# B&R Automation Studio project POM_lab1
Automation Studio 4.5.2.102; technology packages: mappMotion 5.2.1

## Configuration labBR

CPU 4PP065.0571-P74, AutomationRuntime D4.52, Build 4.1.2, Vc V4.52.0, Safety 1.10

### Task classes (Cpu.sw)
```
Cyclic#4:
  Program <- Program.prg
Libraries: McBase, MotorCtrl
```

### Hardware
```
4PP065_0571_P74 : 4PP065.0571-P74 v1.1.2.0
  Connector IF5:
    ActivateDevice = 1
    Mode = Manual
    InternetAddress = 10.0.1.10
    SubnetMask = 255.255.255.0
  ConfigurationID = labBR
  Simulation = 1
```

## Logical view

Binary libraries used (declarations not repeated): operator, runtime, astime, AsIecCon, McBase 5.02.1


### Program Logical/Program (ANSIC)

#### Variables.var
```iecst
VAR
	fb_motor : FB_Motor;
	fb_motor_noreg : FB_Motor;
	fb_regulator : FB_Regulator;
	cnt : USINT;
	speed : REAL;
	enable : BOOL;
END_VAR
```

#### Cyclic.c
```c
#include <bur/plctypes.h>

#ifdef _DEFAULT_INCLUDES
	#include <AsDefault.h>
#endif

void _CYCLIC ProgramCyclic(void)
{
	if(enable) {
		speed = 5;
		cnt++;
	} else {
		speed = 0;
	}
	fb_regulator.e = speed - fb_motor.w;
	fb_motor.u = fb_regulator.u * fb_motor.ke;
	fb_motor_noreg.u = speed * fb_motor_noreg.ke;
	FB_Motor(&fb_motor);
	FB_Motor(&fb_motor_noreg);
	FB_Regulator(&fb_regulator);
}
```

#### Init.c
```c
#include <bur/plctypes.h>

#ifdef _DEFAULT_INCLUDES
	#include <AsDefault.h>
#endif

void _INIT ProgramInit(void)
{
	enable = 0;
	cnt = 0;
	speed = 0;

	fb_motor.dt = 0.02;
	fb_motor.ke = 43.98;
	fb_motor.Tm = 0.173;

	fb_motor_noreg.dt = 0.02;
	fb_motor_noreg.ke = 43.98;
	fb_motor_noreg.Tm = 0.173;

	fb_regulator.dt = 0.02;
	fb_regulator.k_p = 2.174;
	fb_regulator.k_i = 12.56;
	fb_regulator.max_abs_value = 24;
}
```

### Library Logical/MotorCtrl (ANSIC)

#### MotorCtrl.fun - Exported functions and function blocks
```iecst
{REDUND_ERROR} {REDUND_UNREPLICABLE} FUNCTION_BLOCK FB_Integrator (*TODO: Add your comment here*) (*$GROUP=User,$CAT=User,$GROUPICON=User.png,$CATICON=User.png*)
	VAR_INPUT
		in : {REDUND_UNREPLICABLE} REAL;
	END_VAR
	VAR_OUTPUT
		out : {REDUND_UNREPLICABLE} REAL;
	END_VAR
	VAR
		dt : {REDUND_UNREPLICABLE} REAL;
	END_VAR
END_FUNCTION_BLOCK

{REDUND_ERROR} {REDUND_UNREPLICABLE} FUNCTION_BLOCK FB_Motor (*TODO: Add your comment here*) (*$GROUP=User,$CAT=User,$GROUPICON=User.png,$CATICON=User.png*)
	VAR_INPUT
		u : {REDUND_UNREPLICABLE} REAL;
	END_VAR
	VAR_OUTPUT
		w : {REDUND_UNREPLICABLE} REAL;
		phi : {REDUND_UNREPLICABLE} REAL;
	END_VAR
	VAR
		integrator : {REDUND_UNREPLICABLE} FB_Integrator;
		Tm : {REDUND_UNREPLICABLE} REAL;
		ke : {REDUND_UNREPLICABLE} REAL;
		dt : {REDUND_UNREPLICABLE} REAL;
		buf : {REDUND_UNREPLICABLE} REAL;
	END_VAR
END_FUNCTION_BLOCK

{REDUND_ERROR} {REDUND_UNREPLICABLE} FUNCTION_BLOCK FB_Regulator (*TODO: Add your comment here*) (*$GROUP=User,$CAT=User,$GROUPICON=User.png,$CATICON=User.png*)
	VAR_INPUT
		e : {REDUND_UNREPLICABLE} REAL;
	END_VAR
	VAR_OUTPUT
		u : {REDUND_UNREPLICABLE} REAL;
	END_VAR
	VAR
		k_p : {REDUND_UNREPLICABLE} REAL;
		k_i : {REDUND_UNREPLICABLE} REAL;
		integrator : {REDUND_UNREPLICABLE} FB_Integrator;
		iyOld : {REDUND_UNREPLICABLE} REAL;
		max_abs_value : {REDUND_UNREPLICABLE} REAL;
		dt : {REDUND_UNREPLICABLE} REAL;
		buf_up : {REDUND_UNREPLICABLE} REAL;
		buf_down : {REDUND_UNREPLICABLE} REAL;
		sum : {REDUND_UNREPLICABLE} REAL;
	END_VAR
END_FUNCTION_BLOCK
```

#### FB_Integrator.c
```c
#include <bur/plctypes.h>
#ifdef __cplusplus
	extern "C"
	{
#endif
	#include "MotorCtrl.h"
#ifdef __cplusplus
	};
#endif
/* TODO: Add your comment here */
void FB_Integrator(struct FB_Integrator* inst)
{
	inst->dt = 0.02;
	inst->out += inst->dt * inst->in;
}
```

#### FB_Motor.c
```c
#include <bur/plctypes.h>
#ifdef __cplusplus
	extern "C"
	{
#endif
	#include "MotorCtrl.h"
#ifdef __cplusplus
	};
#endif
/* TODO: Add your comment here */
void FB_Motor(struct FB_Motor* inst)
{
	/*TODO: Add your code here*/
	inst->buf = (inst->u * (1/inst->ke) - inst->w)*(1/inst->Tm);

	inst->integrator.in = inst->buf;
	FB_Integrator(&inst->integrator);
	inst->w = inst->integrator.out;

	inst->integrator.in = inst->w;
	FB_Integrator(&inst->integrator);
	inst->phi = inst->integrator.out;
}
```

#### FB_Regulator.c
```c
#include <bur/plctypes.h>
#ifdef __cplusplus
	extern "C"
	{
#endif
	#include "MotorCtrl.h"
#ifdef __cplusplus
	};
#endif
/* TODO: Add your comment here */
void FB_Regulator(struct FB_Regulator* inst)
{
	/*TODO: Add your code here*/
	inst->buf_up = inst->e * inst->k_p;
	if(inst->buf_up > inst->max_abs_value || inst->buf_up < -inst->max_abs_value)
	{
		if (inst->buf_up > 0) {
			inst->buf_up = inst->max_abs_value;
		} else if (inst->buf_up < 0){
			inst->buf_up = -inst->max_abs_value;
		}
	}

	inst->buf_down = inst->e * inst->k_i + inst->iyOld;

	inst->integrator.in = inst->buf_down;
	FB_Integrator(&(inst->integrator));
	inst->buf_down = inst->integrator.out;

	inst->sum = inst->buf_up + inst->buf_down;

	if(inst->sum > inst->max_abs_value || inst->sum < -inst->max_abs_value)
	{
		if (inst->sum > 0) {
			inst->sum = inst->max_abs_value;
		} else if (inst->sum < 0) {
			inst->sum = -inst->max_abs_value;
		}
	}
	inst->u = inst->sum;
	inst->iyOld = inst->u - inst->sum;
}
```

Listed in the project but not available here: Logical/Global.var, Logical/Global.typ, Logical/MotorCtrl/Types.typ, Logical/MotorCtrl/Constants.var
